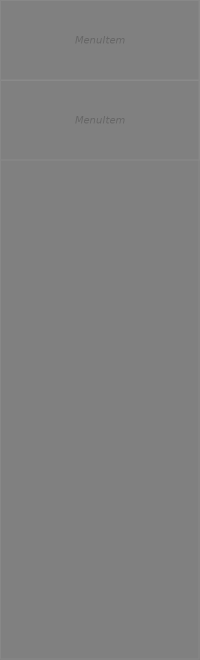
VISUALIZATION Menu  // 200x660
VAR_INPUT
	i_itfVisuMenu : ITF_Visu_Menu;
END_VAR
    Rectangle (0,0 200x660)
    Frame (0,0 200x80)
        shows MenuItem(i_nFrameNumber := 0, i_sText := 'Hoofdmenu', i_itfVisuMenu := i_itfVisuMenu)
    Frame (0,80 200x80)
        shows MenuItem(i_nFrameNumber := 1, i_sText := 'Alarmen', i_itfVisuMenu := i_itfVisuMenu)
END_VISUALIZATION

(* stored: Version 1.1.0.1, ProductVersion 3.1.4026.13
   Visu Menu: Id {9c0d956d-571f-496b-a15d-58fd9429c715} *)
